(*********************************** G.D S.p.A. - Technical Department ***********************************
============= PROGRAM INFO ============
FOLDER:             TBD
MACHINES INVOLVED:  TBD 

============= DESCRIPTION =============

============= REVISIONS ===============
Date		Version	 	Author      	Description             
----------	-------		------------  	--------------------------------------------
2019/04/24 	0000.00	 	M.Grasso		Creation of the PRG

**********************************************************************************************************)
(*$R 
	process_ref:= prc; 
$*)
PROGRAM csp_case_main_safety_drives_SD11000
VAR
	prc:					process;
	prc_path:				STRING;	

	sig:												safety_integrated_group;
	chA_smes_sis:										safety_integrated_series;
	safety_integrated_series_close_dvr_chA: 			BOOL;

	shutdown_chA AT %Q* 								:BOOL := TRUE;
	
END_VAR

_read_var_input();

_objects_manager();

IF NOT objects_running()
THEN
	RETURN;	
END_IF

_read_process_image();

_mode_manager();

//safety_integrated_series_close(chA_smes_sis);

IF  safety_integrated_series_get_mode (chA_smes_sis) = MODE_ABSENT
	OR
	safety_integrated_series_get_mode(chA_smes_sis) = MODE_INACTIVE
	THEN
		shutdown_chA := TRUE;
	ELSE
		shutdown_chA := FALSE;
END_IF

CASE process_get_mode(prc) OF
	MODE_ABSENT,
	MODE_INACTIVE:
		RETURN;
	MODE_TEST:
		;
END_CASE

_set_runtime_properties();

(********************************* BODY *********************************)
IF NOT safety_integrated_group_is_running(sig)
		THEN
			safety_integrated_group_run(sig);
END_IF
safety_integrated_series_close(chA_smes_sis);
safety_integrated_series_close_dvr_chA := safety_integrated_series_is_safely_closed(chA_smes_sis);
(************************************************************************)

_handle_messages();

_write_output();

ACTION _handle_messages:
;
END_ACTION

ACTION _handle_process_test:
;
END_ACTION

ACTION _mode_manager:
IF process_mode_req_is_pending(prc)
THEN
    process_apply_mode_req_first_step(prc);
    CASE process_get_mode(prc) OF
        MODE_TO_ABSENT:
			;
        MODE_TO_INACTIVE:
			;
        MODE_TO_TEST:
			;
        MODE_TO_OPERATIONAL:
			;
    END_CASE
    process_apply_mode_req_second_step(prc);
END_IF
END_ACTION

ACTION _objects_manager:
IF objects_initialization()
THEN
	sub_process_init(
		object_name					:= 'csp_case_main_safety_drives_SD11000.prc', 
		process						:= csp_case_main_safety_drives.prc, 
		CONVERSION_this				:= prc);
		
	prc_path 						:= process_get_path(prc);

	safety_integrated_group_init(
        object_name				:=	CONCAT(prc_path, '_sig'), 
		controller				:=	csp_case_main_safety_interface.SPLC5000_sic,
        process					:=	prc,
        CONVERSION_this			:=	sig);

	(* Channel A SMES series *)
	safety_integrated_series_init(
		object_name				:=	CONCAT(prc_path, '_chA_smes_sis'), 
		_type					:=	SAFETY_INTEGRATED_SERIES_TYPE_NO_RESET,
		discrepancy_active		:=	TRUE,
		forced_open_active		:=	TRUE,
		process					:=	prc,
		CONVERSION_this			:=	chA_smes_sis);

	safety_integrated_series_add_safety_integrated_group(
		group					:=	sig,
		CONVERSION_this			:=	chA_smes_sis);

	safety_integrated_series_add_safety_integrated_series(
		series_active			:=	TRUE,
		series_polarity_direct	:=	TRUE,
		contact					:=	csp_case_main_safety_drives_commonConfiguration.rack_smes_sis, (*Marco : To be checked*)
		CONVERSION_this			:=	chA_smes_sis);
		
END_IF

IF objects_running()
THEN
	process_cycle(prc);
  	safety_integrated_group_cycle(sig);
	safety_integrated_series_cycle(chA_smes_sis);
END_IF
END_ACTION

ACTION _read_process_image:
;
END_ACTION

ACTION _read_var_input:
;
END_ACTION

ACTION _set_runtime_properties:
;
END_ACTION

ACTION _write_output:
;
END_ACTION

END_PROGRAM

(* stored: Version 1.1.0.1, ProductVersion 3.1.4024.3
   POU csp_case_main_safety_drives_SD11000: Id {7ea21db4-c13d-4c3f-bd4d-1c4701f0971f}, SpecialFunc None
   Action _handle_messages: Id {c0329589-594c-440e-a0d4-6e29480fcb6f}
   Action _handle_process_test: Id {268aa9c2-cbb6-47df-9c43-4d1929c479a2}
   Action _mode_manager: Id {2ab6da12-50d4-4567-b848-6878462f95f1}
   Action _objects_manager: Id {7197fd8b-1a42-4814-aed8-231d22b36f33}
   Action _read_process_image: Id {c23dd29b-4d28-4bd5-8d98-aca4b2316d02}
   Action _read_var_input: Id {5d66c9dc-df06-4777-bd6d-fca645689332}
   Action _set_runtime_properties: Id {34e1f3b4-d963-4293-86ec-61317e9a1d19}
   Action _write_output: Id {ba411b98-8146-4a85-bfd5-b344956ed61d} *)
